% RSLogix 500 project 7.3.RSS, saved by version 8.30.00.16 %
PROJECT "7.3"    % processor: Bul.1763 MicroLogix 1100 Series B %

PROGRAM FILES
  LAD 2   6 rungs

DATA FILES
  O0 OUTPUT  4 elements
  I1 INPUT  6 elements
  S2 STATUS  66 elements
  B3 BINARY  1 elements
  T4 TIMER  1 elements
  C5 COUNTER  2 elements
  R6 CONTROL  1 elements
  N7 INTEGER  1 elements
  F8 FLOAT  1 elements

LADDER 2
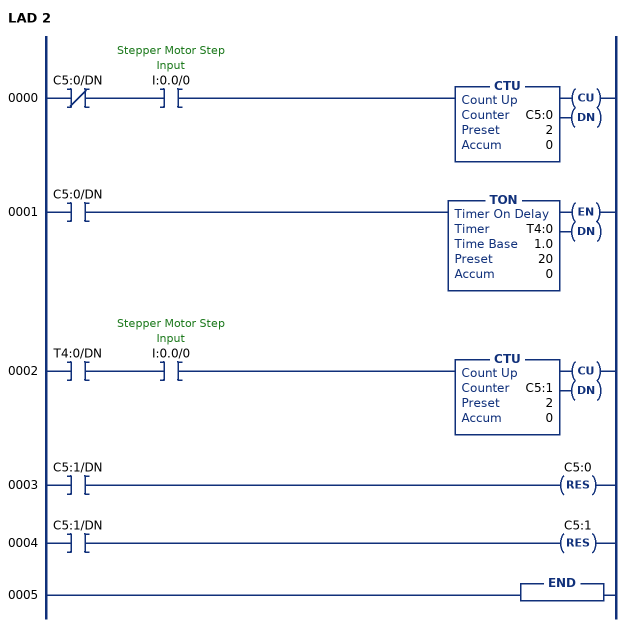
% Rung: 0 %
SOR XIO C5:0/DN XIC I:0.0/0 CTU C5:0 2 0 EOR
%   I:0.0/0  "Stepper Motor Step Input" %
% Rung: 1 %
SOR XIC C5:0/DN TON T4:0 1.0 20 0 EOR
% Rung: 2 %
SOR XIC T4:0/DN XIC I:0.0/0 CTU C5:1 2 0 EOR
%   I:0.0/0  "Stepper Motor Step Input" %
% Rung: 3 %
SOR XIC C5:1/DN RES C5:0 EOR
% Rung: 4 %
SOR XIC C5:1/DN RES C5:1 EOR
% Rung: 5 %
SOR END EOR

DATA TABLE (non-zero values as saved)
DATA T4
% .PRE .ACC %
% T4:0 % 20 0
DATA C5
% .PRE .ACC %
% C5:0 % 2 0
% C5:1 % 2 0
